(* CODESYS project wago_750-658_J1939_demo_v0.0.1.ecp

Project tree, tasks and I/O mapping:
  PFC200_CS_2ETH_RS : 750-8202 PFC200 2ETH RS, WAGO, order no. 0750-8202, version 5.11.1.16
    application Application
      libraries: ; WagoSysErrorBase, * (WAGO); WagoTypesModule_75x_658, 1.6.0.0 (WAGO); Time and Date, 3.5.7.0 (3S - Smart Software Solutions GmbH); WagoTypesCommon, 1.5.2.0 (WAGO); WagoAppCanLayer2, 1.6.0.44 (WAGO); VisuElems, 3.5.11.0 (System)
      task PLC_Task (cyclic, interval t#100ms, priority 14) calls PLC_PRG
      global variables GVL
      program PLC_PRG [ST]
      data type CAN_Data
      program CAN_Gateway [ST]
    DeviceAdapter
    Kbus : Kbus, WAGO, version 1.4.0.2
        unmapped channels: K-BUS diagnostics
      myCANGateway : 0750-0658, WAGO, order no. 0750-0658, version 0.0.0.11
          settings: K-BUS Module slot index = 1; Module attitude = 0750-0658#48
          unmapped channels: _INPUTCHANNEL, _OUTPUTCHANNEL
        DeviceAdapter
    MODBUS
      MODBUS : MODBUS, WAGO, order no. n/a, version 1.1.1.15
    Serial
      COM1 : COM1, WAGO, version 0.0.0.19
  libraries: VisuSymbols, 3.5.10.0 (System); WagoVisuIcons, 1.0.0.8 (WAGO)
  text list GlobalTextList
*)

// PFC200_CS_2ETH_RS/Application/CAN_Data
TYPE CAN_Data :
STRUCT
	ID		: DWORD;
	Data	: ARRAY[0..7]OF BYTE;
END_STRUCT
END_TYPE

// PFC200_CS_2ETH_RS/Application/GVL
{attribute 'qualified_only'}
VAR_GLOBAL
	xFirstScan		: BOOL := TRUE;
	wCanRx29BitAllMsgCounter : WORD;
	myTIme: INT;
END_VAR

// PFC200_CS_2ETH_RS/Application/PLC_PRG
PROGRAM PLC_PRG
VAR
	(* 750-658 CAN Gateway module as J1939 Gateway
	written by: Jesse Cox WAGO USA jesse.cox@wago.com *)
	ftStartScanning		: F_TRIG;
	
	// functional vars
	rtClosePortTrig		: R_TRIG;
	
	// CAN data vars
	BufferIndex			: INT := 0;
	i					: INT;
	myCanData			: ARRAY[0..100] OF CAN_Data;
	myCanMsgCount		: WORD;
	rtReadIntoBuffer	: R_TRIG;
	
	// open block vars
	fbCanOpenPort		: FbCanL2Open;
	xCanPortEnable		: BOOL;
	udiCanPortBaud		: UDINT := 500000;
	dwCanPortFlags		: DWORD := 15;
	xCanPortOpenIsValid	: BOOL;
	xCanPortOpenIsBusy	: BOOL;
	xCanPortOpenError	: BOOL;
	oCanPortOpenStatus	: WagoSysErrorBase.FbResult;
	
	//  close block vars
	fbCanPortClose		: FbCanL2Close;
	xCanPortCloseEnable	: BOOL;
	xCanPortCloseDone	: BOOL;
	xCanPortCloseError	: BOOL;
	xCanPortCloseBusy	: BOOL;
	oCanPortCloseStatus	: WagoSysErrorBase.FbResult;
	
	// Rx vars header
	fbCanRx29Bit				: FbCanRx29BitFrame;
	xCanRx29BitEnable			: BOOL;
	xCanRx29BitBufferEnable		: BOOL;
	dwCanRx29BitID				: DWORD := 16#1CFF0080;  //example header
	xCanRx29BitTrigger			: BOOL;
	xCanRx29BitIsValid			: BOOL;
	xCanRx29BitError			: BOOL;
	xCanRx29BitBusy				: BOOL;
	oCanRx29BitStatus			: WagoSysErrorBase.FbResult;
	wCanRx29BitMsgCounter		: WORD;
	wCanRx29BitFrames			: WORD;
	xCanRx29BitRTR				: BOOL;
	bCanRx29BitBytes			: BYTE;
	aCanRx29BitInBuffer			: ARRAY [1..8] OF BYTE;
	
	// Rx All vars
	fbCanRx29BitAll				: FbCanRx29BitFrameAll;
	xCanRx29BitAllEnable		: BOOL;
	xCanRx29BitAllBufferEnable	: BOOL := TRUE;;
	xCanRx29BitAllTrigger		: BOOL;
	xCanRx29BitAllIsValid		: BOOL;
	xCanRx29BitAllError			: BOOL;
	xCanRx29BitAllBusy			: BOOL;
	oCanRx29BitAllStatus		: WagoSysErrorBase.FbResult;
	wCanRx29BitAllFrames		: WORD;
	xCanRx29BitAllRTR			: BOOL;
	bCanRx29BitAllBytes			: BYTE;
	aCanRx29BitAllInBuffer		: ARRAY [1..8] OF BYTE;
	dwCanRx29BitAllInDataID		: DWORD;
	
	// count valid flags
	rtValid						: R_TRIG;
	wValidJunk					: WORD;
END_VAR

CAN_Gateway();

ftStartScanning(CLK:= GVL.xFirstScan);
IF ftStartScanning.Q THEN
	xCanPortEnable := TRUE;
END_IF

// open the CAN port on the CAn Gateway module
fbCanOpenPort(
	xEnable:= xCanPortEnable, 
	I_Port:= myCANGateway, 
	udiBaudrate:= udiCanPortBaud, 
	dwFlags:= dwCanPortFlags, 
	dwPara:= , 
	xValid=> xCanPortOpenIsValid, 
	xBusy=> xCanPortOpenIsBusy, 
	xError=> xCanPortOpenError, 
	oStatus=> oCanPortOpenStatus);
	
	// enable the read fb when the CAN port is open
	xCanRx29BitAllEnable := xCanPortOpenIsValid;
	
// close the CAN port
fbCanPortClose(
	xExecute:= xCanPortCloseEnable, 
	I_Port:= myCANGateway, 
	xDone=> xCanPortCloseDone, 
	xError=> xCanPortCloseError, 
	xBusy=> xCanPortCloseBusy, 
	oStatus=> oCanPortCloseStatus);	
	
// read the Rx regs
fbCanRx29Bit(
	xEnable:= xCanRx29BitEnable, 
	I_Port:= myCANGateway, 
	xBufferMode:= xCanRx29BitBufferEnable, 
	dwCanId:= dwCanRx29BitID, 
	xRxTrigger:= xCanRx29BitTrigger, 
	xValid=> xCanRx29BitIsValid, 
	xError=> xCanRx29BitError, 
	xBusy=> xCanRx29BitBusy, 
	oStatus=> oCanRx29BitStatus, 
	wCounter=> wCanRx29BitMsgCounter, 
	wFrames=> wCanRx29BitFrames, 
	xRtrFrame=> xCanRx29BitRTR, 
	bRxNBytes=> bCanRx29BitBytes, 
	aRxBuffer=> aCanRx29BitInBuffer);
	
	rtValid(CLK := NOT xCanRx29BitAllIsValid);
	IF rtValid.Q THEN
		wValidJunk := wValidJunk + 1;
	END_IF
	
fbCanRx29BitAll(
	xEnable:= xCanRx29BitAllEnable, 
	I_Port:= myCANGateway, 
	xBufferMode:= xCanRx29BitAllBufferEnable, 
	xRxTrigger:= xCanRx29BitAllTrigger, 
	xValid=> xCanRx29BitAllIsValid, 
	xError=> xCanRx29BitAllError, 
	xBusy=> xCanRx29BitAllBusy, 
	oStatus=> oCanRx29BitAllStatus, 
	wCounter=> GVL.wCanRx29BitAllMsgCounter, 
	wFrames=> wCanRx29BitAllFrames, 
	xRtrFrame=> xCanRx29BitAllRTR, 
	bRxNBytes=> bCanRx29BitAllBytes, 
	aRxBuffer=> aCanRx29BitAllInBuffer, 
	dwRxId=> dwCanRx29BitAllInDataID);
	
	//process the incomming data
	IF xCanRx29BitAllEnable AND ((GVL.wCanRx29BitAllMsgCounter <> myCanMsgCount) OR (wCanRx29BitAllFrames > 0)) THEN
		xCanRx29BitAllTrigger := TRUE;
		myCanMsgCount := GVL.wCanRx29BitAllMsgCounter;
	END_IF
	rtReadIntoBuffer(CLK:= NOT xCanRx29BitAllTrigger);
	IF rtReadIntoBuffer.Q THEN
			myCanData[0].ID := dwCanRx29BitAllInDataID;
			myCanData[0].Data := aCanRx29BitAllInBuffer;
	END_IF

END_PROGRAM

// PFC200_CS_2ETH_RS/Application/CAN_Gateway
PROGRAM CAN_Gateway
VAR
		// variables for configuring CAN Gateway
	fbConfigureCanPort			: FbModuleConfigurationAndStatus;
	xModuleConfigEnable			: BOOL;
	xCanWriteRead				: BOOL;
	xCanSaveValues				: BOOL;
	eCanBitRate					: WagoTypesModule_75x_658.eBitrate := 5;	// 500k
	eMode						: WagoTypesModule_75x_658.eMode := 1;		// transparent mode
	xCan29BitEN					: BOOL;
	xCanSDOEN					: BOOL;
	xCanMBDiagEN				: BOOL;
	typCanConfigData			: WagoTypesModule_75x_658.typFullConfiguration;
	xCanDiagReset				: BOOL;
	xCanCommsReset				: BOOL;
	xCanCheckConfig				: BOOL;
	xCanConfigDone				: BOOL;
	xCanConfigBusy				: BOOL;
	xCanConfigError				: BOOL;
	oCanConfigStatus			: WagoSysErrorBase.FbResult;
	xCanConfigDataMatches		: BOOL;
	eCanDiagErrorCode			: WagoTypesModule_75x_658.eErrorCode;
	bCanDiagChannelNum			: BYTE;
	eCanDiagMode				: WagoTypesModule_75x_658.eDiagQualMode;
	eCanDiagType				: WagoTypesModule_75x_658.eDiagQualType;
	wCanDiagErrorCounter		: WORD;
	wCanDiagWarningCounter		: WORD;
	wCanDiagTotalCounter		: WORD;
	xCanStatusBitModuleError	: BOOL;
	xCanStatusBitRxOverflow		: BOOL;
	xCanStatusBitTxOverflow		: BOOL;
	xCanStatusBitCanError		: BOOL;
	iConfigModuleState			: INT := 0;
	
	// DT vars for error logging
	rtTimeTrigger				: R_TRIG;
	GetDT						: RTCLK.GetDateAndTime;
	xGetDTDone: BOOL;
	xGetDtExecute: BOOL;
	dtHoldDateTime: DATE_AND_TIME;
	dtErrorDateTime: DATE_AND_TIME;
	wMyErrorCounts : WORD;
	myTIme: TIME; 
	
	rtErrorTrig					: R_TRIG;
	wErrorCount					: WORD;
	tTimeRunning				: TIME;
	myStartTime					: TIME;
END_VAR

// configure the CAN module
fbConfigureCanPort(
	I_Port:= myCANGateway, 
	xExecute:= xModuleConfigEnable, 
	xWriteRead:= xCanWriteRead, 
	xSaveValues:= xCanSaveValues, 
	dtTime:= , 
	eBitrate:= eCanBitRate, 
	eMode:= eMode, 
	x29BitEnabled:= xCan29BitEN, 
	xSdoEnabled:= xCanSDOEN, 
	xDiagOverMbx0Enabled:= xCanMBDiagEN, 
	typConfigData:= typCanConfigData, 
	xDiagnosisReset:= xCanDiagReset, 
	xCommunicationReset:= xCanCommsReset, 
	xCheckConfiguration:= xCanCheckConfig, 
	xDone=> xCanConfigDone, 
	xBusy=> xCanConfigBusy, 
	xError=> xCanConfigError, 
	oStatus=> oCanConfigStatus, 
	xDataMatches=> xCanConfigDataMatches, 
	eDiagnosisErrorCode=> eCanDiagErrorCode, 
	bDiagnosisChannelNo=> bCanDiagChannelNum, 
	eDiagnosisMode=> eCanDiagMode, 
	eDiagnosisType=> eCanDiagType, 
	wDiagnosisErrorCounter=> wCanDiagErrorCounter, 
	wDiagnosisWarningCounter=> wCanDiagWarningCounter, 
	wDiagnosisTotalCounter=> wCanDiagTotalCounter, 
	xStatusBitModulError=> xCanStatusBitModuleError, 
	xStatusBitRxOverflow=> xCanStatusBitRxOverflow, 
	xStatusBitTxOverflow=> xCanStatusBitTxOverflow, 
	xStatusBitCanError=> xCanStatusBitCanError);
	
	IF GVL.xFirstScan THEN
		xModuleConfigEnable := TRUE;
		CASE iConfigModuleState OF
		0: // read the settings of the module
			xCan29BitEN := TRUE;
			xCanWriteRead := FALSE;	
			xModuleConfigEnable := TRUE;
			IF xCanConfigDone THEN
				xModuleConfigEnable := FALSE;
				iConfigModuleState := 1;
			END_IF
		1: // write the config
			IF NOT xCanConfigDone THEN
				xCanWriteRead := TRUE;	
			xModuleConfigEnable := TRUE;
			ELSE
				xModuleConfigEnable := FALSE;
				iConfigModuleState := 2;
			END_IF
		2: // verify match
			xModuleConfigEnable := FALSE;
			xCanCheckConfig := TRUE;
			IF xCanConfigDataMatches THEN
				GVL.xFirstScan := FALSE;
				myStartTime := TIME();
				iConfigModuleState := 0;
			END_IF
		END_CASE
	END_IF
	
	rtTimeTrigger(CLK:= xCanStatusBitModuleError);
	IF rtTimeTrigger.Q THEN
		xGetDtExecute := TRUE;
		dtErrorDateTime := dtHoldDateTime;
		wMyErrorCounts := GVL.wCanRx29BitAllMsgCounter;
	END_IF
	GetDT(
	xExecute:= xGetDtExecute, 
	xDone=> xGetDTDone, 
	xBusy=> , 
	xError=> , 
	eError=> , 
	dtDateAndTime=> dtHoldDateTime, 
	eTimezone=> );
	
	myTIme := TIME() - myStartTime;
	rtErrorTrig(CLK:= xCanStatusBitModuleError);
	IF rtErrorTrig.Q THEN
		wErrorCount := wErrorCount + 1;
	END_IF

END_PROGRAM
